Yaskawa INFORM job: X2_NOWY.JBI

/JOB
//NAME X2_NOWY
//POS
///NPOS 60,60,60,5,0,0
///TOOL 0
///POSTYPE PULSE
///PULSE
C00000=-3270,-119374,-120744,349,28960,-82703
C00001=89062,-116132,-100192,547,17977,-82798
C00002=128610,-85662,-90756,-15107,33359,-75826
C00003=123876,-80225,-87696,-8948,33562,-78713
C00004=128929,-77617,-86369,-14950,34802,-75943
C00005=128929,-77698,-85716,-15117,34375,-75851
C00006=128929,-77681,-85864,-15079,34472,-75871
C00007=128766,-74686,-84474,-14633,35105,-76097
C00008=129052,-79841,-87430,-15280,34354,-75772
C00009=146845,-41555,-81100,23854,45661,-87406
C00010=146839,-41400,-81183,23823,45788,-87374
C00011=146839,-41975,-80694,24057,45240,-87525
C00012=146839,-41846,-80806,24003,45364,-87490
C00013=146435,-39406,-79308,24256,45771,-87555
C00014=146839,-41846,-80806,24003,45364,-87490
C00015=145883,-63774,-98880,7542,46700,-84601
C00016=155389,-119793,-121385,-2447,31472,-80379
C00017=102037,-133341,-129837,-2447,31472,-80379
C00018=113521,-70304,-99610,-13723,42507,-75289
C00019=113576,-69044,-98954,-13718,42751,-75304
C00020=113576,-69643,-98389,-13887,42113,-75201
C00021=113576,-69532,-98497,-13855,42233,-75221
C00022=113703,-66519,-97031,-13821,42882,-75268
C00023=113576,-69215,-98799,-13765,42572,-75276
C00024=116385,-35976,-77484,-50912,59283,-62708
C00025=116385,-35838,-77595,-50848,59373,-62765
C00026=116385,-36432,-77104,-51124,58981,-62518
C00027=116365,-37033,-77677,-51091,59000,-62539
C00028=116427,-34715,-76197,-51001,59211,-62640
C00029=116365,-37033,-77677,-51091,59000,-62539
C00030=117692,-43924,-75065,-61492,51873,-58717
C00031=118714,-28601,-66381,-64093,60579,-60179
C00032=115289,-24898,-63546,-64080,60206,-60356
C00033=114902,-26070,-64609,-63051,59070,-60714
C00034=127850,-26661,-63451,-72108,65262,-58732
C00035=130557,-33924,-68329,-73549,66718,-58095
C00036=106572,-58848,-93942,-15426,45804,-80121
C00037=106805,-57523,-92479,-15708,45631,-79993
C00038=102131,-55362,-91307,-11025,45331,-81929
C00039=108857,-71296,-101220,-18205,44385,-78853
C00040=110435,-82200,-106133,-1038,40006,-86002
C00041=110257,-62003,-97964,-607,48269,-86053
C00042=105614,-60279,-97081,3756,48691,-87855
C00043=103782,-78639,-107364,5746,45692,-88747
C00044=132684,-130914,-127982,-52253,49571,-61610
C00045=139278,-129792,-110794,-83567,32161,-45718
C00046=120590,-62989,-101418,-16330,54617,-61245
C00047=125691,-55599,-96750,-25151,57981,-57710
C00048=123873,-57083,-96193,-26483,55772,-59137
C00049=127522,-66713,-102028,-29694,55636,-57651
C00050=107332,-64864,-101121,24429,54104,-80168
C00051=108176,-57800,-96477,23538,54601,-79719
C00052=114103,-61547,-97621,19306,51151,-78126
C00053=113976,-63835,-99856,19057,52338,-77968
C00054=99110,-36748,-75475,61977,67040,-86750
C00055=102032,-35871,-73292,63729,66095,-86717
C00056=95054,-53921,-86066,55693,56200,-84395
C00057=78339,-85415,-97950,74258,61103,-88238
C00058=70048,-95947,-100914,80606,65818,-89400
C00059=-3270,-119374,-120744,349,28960,-82703
BC00000=132367,523905,620572
BC00001=246832,523905,238784
BC00002=314526,523905,238784
BC00003=314526,523905,238784
BC00004=314526,523905,238784
BC00005=314526,523905,238784
BC00006=314526,523905,238784
BC00007=314526,523905,238784
BC00008=314526,523905,238784
BC00009=380619,523905,111536
BC00010=380618,523904,111533
BC00011=380618,523904,111533
BC00012=380618,523904,111533
BC00013=380618,523904,111533
BC00014=380618,523904,111533
BC00015=380618,523904,111533
BC00016=380618,523904,111533
BC00017=89188,526512,111533
BC00018=89188,526512,111533
BC00019=89188,526512,111533
BC00020=89188,526512,111533
BC00021=89188,526512,111533
BC00022=89188,526512,111533
BC00023=89188,526512,111533
BC00024=89188,526512,111533
BC00025=89188,526512,111533
BC00026=89188,526512,111533
BC00027=89188,526512,111533
BC00028=89188,526512,111533
BC00029=89188,526512,111533
BC00030=89188,526512,111533
BC00031=89188,526512,111533
BC00032=89189,526511,111532
BC00033=89188,526512,111533
BC00034=89188,526512,111533
BC00035=89188,526512,111533
BC00036=89188,526512,111533
BC00037=89188,526512,111533
BC00038=89188,526512,111533
BC00039=89188,526512,111533
BC00040=89188,526512,111533
BC00041=89188,526512,111533
BC00042=89188,526512,111533
BC00043=89188,526512,111533
BC00044=89188,524556,111533
BC00045=294788,524556,111533
BC00046=294788,524556,111533
BC00047=294788,524556,111533
BC00048=294788,524556,111533
BC00049=294788,524556,111533
BC00050=294788,524556,111533
BC00051=294788,524556,111533
BC00052=294788,524556,111533
BC00053=294788,524556,111533
BC00054=294788,524556,111533
BC00055=294788,524556,111531
BC00056=294788,524556,111531
BC00057=294788,524556,111531
BC00058=294788,524556,111531
BC00059=132367,523905,620572
EC00000=77843,371283
EC00001=77843,371283
EC00002=77843,371283
EC00003=77843,371283
EC00004=77843,371283
EC00005=77843,371283
EC00006=77843,371283
EC00007=77843,371283
EC00008=77843,371283
EC00009=77843,371283
EC00010=77844,371284
EC00011=77844,371284
EC00012=77844,371284
EC00013=77844,371284
EC00014=77844,371284
EC00015=77844,371284
EC00016=77844,371284
EC00017=77844,371284
EC00018=77844,371284
EC00019=77844,371284
EC00020=77844,371284
EC00021=77844,371284
EC00022=77844,371284
EC00023=77844,371284
EC00024=77844,371284
EC00025=77844,371284
EC00026=77844,371284
EC00027=77844,371284
EC00028=77844,371284
EC00029=77844,371284
EC00030=77844,371284
EC00031=77844,371284
EC00032=77845,371284
EC00033=77844,371284
EC00034=77844,371284
EC00035=77844,371284
EC00036=77844,371284
EC00037=77844,371284
EC00038=77844,371284
EC00039=77844,371284
EC00040=77844,371284
EC00041=77844,371284
EC00042=77844,371284
EC00043=77844,371284
EC00044=77844,371284
EC00045=77844,371284
EC00046=77844,371284
EC00047=77844,371284
EC00048=77844,371284
EC00049=77844,371284
EC00050=77844,371284
EC00051=77844,371284
EC00052=77844,371284
EC00053=77844,371284
EC00054=77844,371284
EC00055=77844,371284
EC00056=77844,371284
EC00057=77844,371284
EC00058=77844,371284
EC00059=77843,371283
///POSTYPE BASE
///RECTAN
///RCONF 0,0,0,0,1,0,0,0,0,0,0,0,0,0,0,0,0,0,0,0,0,0,0,0
P00006=2.006,1.622,-0.565,0.0000,0.0000,0.0000
///RCONF 0,0,0,0,0,0,0,0,0,0,0,0,0,0,0,0,0,0,0,0,0,0,0,0
P00031=-0.170,0.039,-0.647,0.0000,0.0000,0.0000
P00032=-0.423,0.157,3.222,0.0000,0.0000,0.0000
P00033=0.854,-1.099,3.047,0.0000,0.0000,0.0000
///RCONF 0,0,0,0,1,0,0,0,0,0,0,0,0,0,0,0,0,0,0,0,0,0,0,0
P00034=-8.151,9.743,-4.393,0.0000,0.0000,0.0000
//INST
///DATE 2024/12/17 23:44
///COMM BRAKUJACE SPOINY
///ATTR SC,RW
///GROUP1 RB1,BS1
///GROUP2 ST1
NOP
MOVJ C00000 BC00000 VJ=100.00  +MOVJ EC00000 VJ=100.00
MOVJ C00001 BC00001 VJ=100.00  +MOVJ EC00001 VJ=100.00
MOVJ C00002 BC00002 VJ=40.00  +MOVJ EC00002 VJ=100.00
SMOVL C00003 BC00003 V=150.0  +MOVJ EC00003
SMOVL C00004 BC00004 V=166.7  +MOVJ EC00004
SREFP 3 C00005 BC00005  +REFP EC00005
CALL JOB:SEARCH-R1-S13D
SET P031 P006
SFTON3D P031
SMOVL C00006 BC00006 V=166.7  +MOVJ EC00006
SREFP 3 C00007 BC00007  +REFP EC00007
CALL JOB:SEARCH-R1-S13D
SET P031 P006
SFTON3D P031
SMOVL C00008 BC00008 V=150.0  +MOVJ EC00008
SFTOF3D
SMOVL C00009 BC00009 V=250.0  +MOVJ EC00009
SMOVL C00010 BC00010 V=166.7  +MOVJ EC00010
SREFP 3 C00011 BC00011  +REFP EC00011
CALL JOB:SEARCH-R1-S13D
SET P032 P006
SFTON3D P032
SMOVL C00012 BC00012 V=166.7  +MOVJ EC00012
SREFP 3 C00013 BC00013  +REFP EC00013
CALL JOB:SEARCH-R1-S13D
SET P032 P006
SFTON3D P032
SMOVL C00014 BC00014 V=166.7  +MOVJ EC00014
SFTOF3D
SMOVL C00015 BC00015 V=166.7  +MOVJ EC00015
SMOVL C00016 BC00016 V=333.3  +MOVJ EC00016
SMOVL C00017 BC00017 V=666.7  +MOVJ EC00017
SMOVL C00018 BC00018 V=333.3  +MOVJ EC00018
SMOVL C00019 BC00019 V=166.7  +MOVJ EC00019
SREFP 3 C00020 BC00020  +REFP EC00020
CALL JOB:SEARCH-R1-S13D
SET P033 P006
SFTON3D P033
SMOVL C00021 BC00021 V=166.7  +MOVJ EC00021
SREFP 3 C00022 BC00022  +REFP EC00022
CALL JOB:SEARCH-R1-S13D
SET P033 P006
SFTON3D P033
SMOVL C00023 BC00023 V=166.7  +MOVJ EC00023
SFTOF3D
SMOVL C00024 BC00024 V=333.3  +MOVJ EC00024
SMOVL C00025 BC00025 V=166.7  +MOVJ EC00025
SREFP 3 C00026 BC00026  +REFP EC00026
CALL JOB:SEARCH-R1-S13D
SET P034 P006
SFTON3D P034
SMOVL C00027 BC00027 V=166.7  +MOVJ EC00027
SREFP 3 C00028 BC00028  +REFP EC00028
CALL JOB:SEARCH-R1-S13D
SET P034 P006
SFTON3D P034
SMOVL C00029 BC00029 V=166.7  +MOVJ EC00029
SMOVL C00030 BC00030 V=150.0  +MOVJ EC00030
MACRO1 MJ#(0) ARGF14
SMOVL C00031 BC00031 V=333.3  +MOVJ EC00031
ARCON
SMOVL C00032 BC00032 V=10.0  +MOVJ EC00032
ARCOF
SMOVL C00033 BC00033 V=166.7  +MOVJ EC00033
SMOVL C00034 BC00034 V=166.7  +MOVJ EC00034
SMOVL C00035 BC00035 V=166.7  +MOVJ EC00035
SMOVL C00036 BC00036 V=166.7  +MOVJ EC00036
SMOVL C00037 BC00037 V=166.7  +MOVJ EC00037
ARCON
SMOVL C00038 BC00038 V=10.0  +MOVJ EC00038
ARCOF
SMOVL C00039 BC00039 V=166.7  +MOVJ EC00039
SFTOF3D
SMOVL C00040 BC00040 V=166.7  +MOVJ EC00040
SFTON3D P033
SMOVL C00041 BC00041 V=166.7  +MOVJ EC00041
ARCON
SMOVL C00042 BC00042 V=10.0  +MOVJ EC00042
ARCOF
SMOVL C00043 BC00043 V=250.0  +MOVJ EC00043
SFTOF3D
SMOVL C00044 BC00044 V=666.7  +MOVJ EC00044
SMOVL C00045 BC00045 V=666.7  +MOVJ EC00045
SMOVL C00046 BC00046 V=333.3  +MOVJ EC00046
SFTON3D P031
SMOVL C00047 BC00047 V=166.7  +MOVJ EC00047
ARCON
SMOVL C00048 BC00048 V=10.0  +MOVJ EC00048
ARCOF
SMOVL C00049 BC00049 V=166.7  +MOVJ EC00049
SMOVL C00050 BC00050 V=166.7  +MOVJ EC00050
SFTON3D P032
SMOVL C00051 BC00051 V=166.7  +MOVJ EC00051
ARCON
SMOVL C00052 BC00052 V=10.0  +MOVJ EC00052
ARCOF
SMOVL C00053 BC00053 V=133.3  +MOVJ EC00053
SMOVL C00054 BC00054 V=250.0  +MOVJ EC00054
ARCON
SMOVL C00055 BC00055 V=10.0  +MOVJ EC00055
ARCOF
SMOVL C00056 BC00056 V=333.3  +MOVJ EC00056
SFTOF3D
SMOVL C00057 BC00057 V=666.7  +MOVJ EC00057
MOVJ C00058 BC00058 VJ=100.00  +MOVJ EC00058 VJ=100.00
MOVJ C00059 BC00059 VJ=100.00  +MOVJ EC00059 VJ=100.00
END
